# EPICS alarm handler configuration: alh_files/mgnt_bsyA_lgps.alhConfig
GROUP NULL LGPS:BSYA:MG01
   $COMMAND edm -x -eolc -noedit mgnt_bsy0_main.edl
$ALIAS LGPS
$GUIDANCE
BSYA LGPS
   Group Name: LGPS:BSYA:MG01
   Summary PV:  LGPS:BSYA:MG01:STATSUMY
$END

GROUP LGPS:BSYA:MG01  LGPS:AB01:1100
CHANNEL    LGPS:AB01:1100    LGPS:AB01:1100:BACTAPV   -----
   $FORCEPV LGPS:AB01:1100:BACTAPVSV -DATL 1 0
